{attribute 'qualified_only'}
{attribute 'strict'}
TYPE E_ValveResetState :
(
	Res_Idle 		:= 0,
	Res_Closed		:= 1,
	Res_Open		:= 2
);
END_TYPE

(* stored: Version 1.1.0.1, ProductVersion 3.1.4022.16
   EnumerationTextList E_ValveResetState: Id {431c2c59-1f9a-4043-a18b-13d165d5ba08} *)
